PROGRAM CraneSimulation
VAR
	fTime : LREAL; 	
	bRunning : BOOL;
	fPositionAutoMode : LREAL; 
	fInitialPosition : LREAL; 
	fInitialVelocity : LREAL;
	eStatus : E_CraneStatus;
	eMode : E_CraneMode;
	aPistonEndStopMsg : ARRAY [0..2] OF STRING := ['End Stop not active', 'Piston has reached upper End Stop', 'Piston has reached Lower End Stop'];
 	fPressureEng : REAL;
	fFlowEng : REAL;
	fPressureBar : LREAL := 60;
	fFlowLmin : LREAL := 20;
	bPistonMaxNewValue : BOOL;
	fMaxPistonPosition : LREAL;
END_VAR

IF Inputs.bStartSimulation AND Inputs.bAutoMode  THEN
	fTime := fTime + Parameters.fCyclicTime;
ELSE
	fTime := 0; 	
END_IF

IF fTime > 0 AND Inputs.bAutoMode THEN 
	bRunning := TRUE;
ELSE
	bRunning := FALSE;
END_IF

fPositionAutoMode := Inputs.fCylinderVelocityReference * 1/2*(fTime*fTime) + fInitialVelocity * fTime + fInitialPosition;

// added max/min outout value to avoid to large output for visualization
IF fPositionAutoMode >= Parameters.stPistonRange.fPistonPosMax THEN
	fPositionAutoMode := Parameters.stPistonRange.fPistonPosMax;	
ELSIF fPositionAutoMode <= Parameters.stPistonRange.fPistonPosMin  THEN
	fPositionAutoMode := Parameters.stPistonRange.fPistonPosMin; 
ELSE	
	fPositionAutoMode := fPositionAutoMode;
END_IF

IF Inputs.bAutoMode THEN
	Outputs.fCylinderPosition := fPositionAutoMode;
ELSE
	Outputs.fCylinderPosition := Inputs.fManualCylinderPositionReference;	
END_IF


Outputs.bSimulationRunning := bRunning;  
Outputs.fSimulationTime := fTime; 
Outputs.fCylinderVelocity := Inputs.fCylinderVelocityReference;
Outputs.pt1_y := LREAL_TO_INT(Outputs.fCylinderPosition * Parameters.fPistonScale);

//status
IF inputs.bEnableSimulation THEN
	eStatus := E_CraneStatus.Ready;
ELSE
	eStatus := E_CraneStatus.Faulty;
END_IF

IF inputs.bStartSimulation THEN
	eStatus := E_CraneStatus.Starting;
END_IF

IF Outputs.bSimulationRunning THEN
	eStatus := E_CraneStatus.Running;
END_IF

//mode
IF inputs.bAutoMode THEN
	eMode := E_CraneMode.Auto;
ELSE
	eMode := E_CraneMode.Manual;
END_IF

//Logic for pistonStops
IF Outputs.fCylinderPosition <= Parameters.stPistonRange.fPistonPosMin THEN
	Outputs.bPistonLowerEndStop := TRUE;
	Outputs.bPistonUpperEndStop := FALSE;
	HMI.sPistonEndStopMessages := aPistonEndStopMsg[2];
	
ELSIF Outputs.fCylinderPosition >= Parameters.stPistonRange.fPistonPosMax THEN
	Outputs.bPistonLowerEndStop := FALSE;
	Outputs.bPistonUpperEndStop := TRUE;
	HMI.sPistonEndStopMessages := aPistonEndStopMsg[1];

ELSE
	Outputs.bPistonLowerEndStop := FALSE;
	Outputs.bPistonUpperEndStop := FALSE;
	HMI.sPistonEndStopMessages := aPistonEndStopMsg[0];
END_IF

//unit conversions

fPressureEng := LREAL_TO_REAL (F_BarToEng(fBar := fPressureBar));
fFlowEng := LREAL_TO_REAL (F_LminToEng(fLminFlow := fFlowLmin));

//Piston stroke

F_UpdateParametersByReference(
	bSetNewValue := bPistonMaxNewValue,
	fMaxPistonStroke := fMaxPistonPosition,
	paramCylinderPiston := Parameters.stPistonRange
);

END_PROGRAM

(* stored: Version 1.1.0.1, ProductVersion 3.1.4024.10
   POU CraneSimulation: Id {c255987f-7a58-4573-9ac9-545c12e8d4a5}, SpecialFunc None *)
